// TIA Portal V17 export
// export: Created 2025-03-13T10:30:31.2703553Z, ExportSetting WithDefaults, DisplayName Totally Integrated Automation Portal, DisplayVersion V17 Update 8, DisplayName TIA Portal Openness, DisplayVersion V17 Update 8, DisplayName TIA Portal Version Control Interface, DisplayVersion V17, DisplayName SINAMICS Startdrive Advanced, DisplayVersion V17 SP2, DisplayName SINAMICS Startdrive G110M, G120, G120C, G120D, G120P, G115D, DisplayVersion V17 SP2, DisplayName SINAMICS Startdrive G130, G150, S120, S150, SINAMICS MV, S210, DisplayVersion V17 SP2, DisplayName STEP 7 Professional, DisplayVersion V17 Update 8, DisplayName SINUMERIK ONE STEP 7 Toolbox, DisplayVersion V17 Update 12, DisplayName SINUMERIK 840D sl STEP 7 Toolbox, DisplayVersion V17 Update 12, DisplayName STEP 7 Safety, DisplayVersion V17 Update 6, DisplayName WinCC Advanced, DisplayVersion V17 Update 8
DATA_BLOCK "DB2440_GLOBAL_DATA"   // DB2440
{ S7_Optimized_Access := 'FALSE'; DB_Accessible_From_OPC_UA := 'FALSE' }
AUTHOR : ETXETAR
NAME : XFLX-DUO
VERSION : 1.0
// stored: AutoNumber false, DBAccessibleFromOPCUA false, DBAccessibleFromWebserver true, IsOnlyStoredInLoadMemory false, IsWriteProtectedInAS false
   VAR RETAIN
      GLOBAL_DATA { S7_SetPoint := 'True'} : "GLOBAL_DATA_CLADDING";
      AXIS_MANAGEMENT { S7_SetPoint := 'True'} : "AXIS_MANAGEMENT";
      OPTIONS : Struct
         PHD : Bool;   // PART HANDLING DEVICE OPTION
         LIFTING_SLIDE : Bool;   // LIFTING SLIDE OPTION
         X_FLEX_DUO : Bool;   // X FLEX DUO OPTION
         X_FLEX_TWIN : Bool;   // X FLEX TWIN OPTION
         BYPASS_Z11 : Bool;   // BYPASS Z11 OPTION
         BYPASS_Z12 : Bool;   // BYPASS Z12 OPTION
         BYPASS_Z21 : Bool;   // BYPASS Z21 OPTION
         BYPASS_Z22 : Bool;   // BYPASS Z22 OPTION
         NO_MAGAZINE : Bool;   // MACHINE WITHOUT MAGAZINE / NO MAGAZINE OPTION
         UNIT_02_AVAILABLE : Bool;   // INDEPENDENT Z AXES OPTION
      END_STRUCT;
      TIMER_DELAY_ANY_CYCLE_RUN { S7_SetPoint := 'True'} : TOF_TIME;
      TIMER_DELAY_ANY_CYCLE_RUN_UNIT_01 { S7_SetPoint := 'True'} : TOF_TIME;
      TIMER_DELAY_ANY_CYCLE_RUN_UNIT_02 { S7_SetPoint := 'True'} : TOF_TIME;
      TIMER_DELAY_ANY_CYCLE_RUN_UNIT_03 { S7_SetPoint := 'True'} : TOF_TIME;
      TIMER_DELAY_ANY_CYCLE_RUN_HOPPER_UNIT_01 { S7_SetPoint := 'True'} : TOF_TIME;
      TIMER_DELAY_ANY_CYCLE_RUN_HOPPER_UNIT_02 { S7_SetPoint := 'True'} : TOF_TIME;
      TIMER_DELAY_RESET_FULL_DEPTH_U1_F1 { S7_SetPoint := 'True'} : TON_TIME;
      TIMER_DELAY_RESET_FULL_DEPTH_U1_F2 { S7_SetPoint := 'True'} : TON_TIME;
      TIMER_DELAY_RESET_FULL_DEPTH_U1_F3 { S7_SetPoint := 'True'} : TON_TIME;
      TIMER_DELAY_RESET_FULL_DEPTH_U1_F4 { S7_SetPoint := 'True'} : TON_TIME;
      TIMER_DELAY_RESET_FULL_DEPTH_U2_F1 { S7_SetPoint := 'True'} : TON_TIME;
      TIMER_DELAY_RESET_FULL_DEPTH_U2_F2 { S7_SetPoint := 'True'} : TON_TIME;
      TIMER_DELAY_RESET_FULL_DEPTH_U2_F3 { S7_SetPoint := 'True'} : TON_TIME;
      TIMER_DELAY_RESET_FULL_DEPTH_U2_F4 { S7_SetPoint := 'True'} : TON_TIME;
   END_VAR
BEGIN
   TIMER_DELAY_ANY_CYCLE_RUN.PT := T#500ms;
   TIMER_DELAY_ANY_CYCLE_RUN_UNIT_01.PT := T#500ms;
   TIMER_DELAY_ANY_CYCLE_RUN_UNIT_02.PT := T#500ms;
   TIMER_DELAY_ANY_CYCLE_RUN_UNIT_03.PT := T#500ms;
   TIMER_DELAY_ANY_CYCLE_RUN_HOPPER_UNIT_01.PT := T#500ms;
   TIMER_DELAY_ANY_CYCLE_RUN_HOPPER_UNIT_02.PT := T#500ms;
   TIMER_DELAY_RESET_FULL_DEPTH_U1_F1.PT := T#10s;
   TIMER_DELAY_RESET_FULL_DEPTH_U1_F2.PT := T#10s;
   TIMER_DELAY_RESET_FULL_DEPTH_U1_F3.PT := T#10s;
   TIMER_DELAY_RESET_FULL_DEPTH_U1_F4.PT := T#10s;
   TIMER_DELAY_RESET_FULL_DEPTH_U2_F1.PT := T#10s;
   TIMER_DELAY_RESET_FULL_DEPTH_U2_F2.PT := T#10s;
   TIMER_DELAY_RESET_FULL_DEPTH_U2_F3.PT := T#10s;
   TIMER_DELAY_RESET_FULL_DEPTH_U2_F4.PT := T#10s;
END_DATA_BLOCK
